FUNCTION_BLOCK FB_LinkedList_Test EXTENDS FB_TestSuite
VAR
END_VAR

NewListHasLength0();
isEmptyReturnsTrueOnEmptyList();
AddFirstNode();
AddMultipleNodesSameType();
AddMultipleNodesDifferentTypes();
InsertAfterSuccessfully();
RemoveNodeSuccessfully();

METHOD AddFirstNode
VAR
	fbLinkedList : FB_LinkedList;
	
	value : INT := 1;
	getValue : INT;
	
	Actual1 : BOOL;
	Actual2 : UINT;
	Actual3 : INT;
	
	Expected1 : BOOL := FALSE;
	Expected2 : UINT := 1;
	Expected3 : INT := 1;
END_VAR
TEST('AddFirstNode');

fbLinkedList.addValue(value);

Actual1 := fbLinkedList.isEmpty();
AssertEquals(Expected := Expected1, Actual := Actual1, Message := 'isEmpty returns true after adding an item to the list');

Actual2 := fbLinkedList.Length;
AssertEquals(Expected := Expected2, Actual := Actual2, Message := 'Length is not equal to 1 after adding 1 node');

fbLinkedList.getValue(0,getValue);
Actual3 := getValue;
AssertEquals(Expected := Expected3, Actual := Actual3, Message := 'getValue did not return the expected value');

TEST_FINISHED();
END_METHOD

METHOD AddMultipleNodesDifferentTypes
VAR
	fbLinkedList: FB_LinkedList;
	
	intValue 		: INT 		:= 33;
	realValue 		: REAL		:= 3.123;
	stringValue 	: STRING 	:= 'Hello world!';
	
	getInt : INT;
	getReal : REAL;
	getString : STRING;
	
	actualint : INT;
	actualReal : REAL;
	actualString : STRING;
END_VAR
TEST('AddMultipleNodesDifferentTypes');

fbLinkedList.addValue(intValue);
fbLinkedList.addValue(realValue);
fbLinkedList.addValue(stringValue);

fbLinkedList.getValue(0,getInt);
actualInt :=  getInt;
fbLinkedList.getValue(1, getReal);
actualReal := getReal;
fbLinkedList.getValue(2,getString);
actualString := getString;

AssertEquals_INT(expected := intValue, actual := actualInt, message := 'Position 0 was unexpected value');
AssertEquals_REAL(expected := realValue, actual := actualReal, delta := 0.01, message := 'Position 1 was unexpected value');
AssertEquals_STRING(expected := stringValue, actual := actualString, message := 'Position 2 was unexpceted value');

TEST_FINISHED();
END_METHOD

METHOD AddMultipleNodesSameType
VAR
	fbLinkedList : FB_LinkedList;
	intArray : ARRAY [0..4] OF INT := [1,2,3,4,5];
	i : INT;
	Actual: INT;
	ActualArr: INT;
	Expected: INT := 5;
	ExpectedArr: INT;
END_VAR
TEST('AddMultipleNodesSameType');

FOR i := 0 TO 4 DO
	fbLinkedList.addValue(intArray[i]);
END_FOR

Actual := fbLinkedList.Length;
AssertEquals(Expected := Expected, Actual := Actual, Message := 'Length not equal to 5 after adding 5 nodes');

FOR i := 0 TO 4 DO 
	fbLinkedList.getValue(i, ActualArr);
	ExpectedArr := intArray[i];
	AssertEquals(Expected := ExpectedArr, 
				 Actual := ActualArr, 
				 Message := CONCAT('Index ',CONCAT( INT_TO_STRING(i), CONCAT( ', expected ', CONCAT(INT_TO_STRING(ExpectedArr), CONCAT(', got ', INT_TO_STRING(ActualArr)))))));  
END_FOR

TEST_FINISHED();
END_METHOD

METHOD InsertAfterSuccessfully
VAR
	fbLinkedList : FB_LinkedList;
	initArray : ARRAY [0..4] OF INT := [1,2,3,4,5];
	i : INT;
	
	value : INT := 6;
	
	expectedArray : ARRAY [0..5] OF INT := [1,2,3,4,6,5];
	
	actual : INT;
	expected : INT;
END_VAR
TEST('InsertAfterSuccessfully');

FOR i := 0 TO 4 DO
	fbLinkedList.addValue(initArray[i]);
END_FOR

fbLinkedList.insertAfter(value, 3);

FOR i := 0 TO 4 DO 
	fbLinkedList.getValue(i, actual);
	expected := expectedArray[i];
	AssertEquals(Expected := Expected, Actual := Actual, Message := CONCAT('Index ', CONCAT(INT_TO_STRING(i), ' is not the expcted value'))); 
END_FOR

TEST_FINISHED();
END_METHOD

METHOD isEmptyReturnsTrueOnEmptyList
VAR
	fbLinkedList : FB_LinkedList;
	Expected : BOOL := TRUE;
	Actual: BOOL;
END_VAR
TEST('isEmptyReturnsTrueOnEmptyList');

Actual := fbLinkedList.isEmpty();

AssertEquals(Expected := Expected,
			 Actual := Actual,
			 Message := 'isEmpty() evaluates false on new linked list');
			 
TEST_FINISHED();
END_METHOD

METHOD NewListHasLength0
VAR
	LinkedList : FB_LinkedList;
	Result : UINT;
	ExpectedLength : UINT := 0;
END_VAR
TEST('NewListHasLength0');

Result := LinkedList.Length;

AssertEquals(Expected := ExpectedLength,
			Actual := Result,
			Message := 'New list is not empty');
			
			
	

TEST_FINISHED();
END_METHOD

METHOD RemoveNodeSuccessfully
VAR
	fbLinkedList : FB_LinkedList;
	initArray : ARRAY [0..4] OF INT := [1,2,3,4,5];
	i : INT;
	
	expectedArray : ARRAY [0..3] OF INT := [1,2,4,5];
	
	actual : INT;
	expected : INT;
END_VAR
TEST('RemoveNodeSuccessfully');

FOR i := 0 TO 4 DO
	fbLinkedList.addValue(initArray[i]);
END_FOR

fbLinkedList.remove(2);

FOR i := 0 TO 4 DO 
	fbLinkedList.getValue(i, actual);
	expected := expectedArray[i];
	AssertEquals(Expected := Expected, Actual := Actual, Message := CONCAT('Index ', CONCAT(INT_TO_STRING(i), ' is not the expcted value'))); 
END_FOR

TEST_FINISHED();
END_METHOD

END_FUNCTION_BLOCK

(* stored: Version 1.1.0.1
   POU FB_LinkedList_Test: Id {3d9ebd70-657f-405b-b31e-010edd5810ad}, SpecialFunc None
   Method AddFirstNode: Id {02c4374d-54e1-4c6d-a171-b7c57fceb053}
   Method AddMultipleNodesDifferentTypes: Id {cd39a802-fd8b-4efc-aea3-df781ae0ac28}
   Method AddMultipleNodesSameType: Id {8224b165-2d73-4654-aee9-e1a98ae56ad8}
   Method InsertAfterSuccessfully: Id {b32a3f05-51de-4288-b235-a3ce606ef510}
   Method isEmptyReturnsTrueOnEmptyList: Id {f9b33b21-fb22-40ad-9f99-3999b9a82141}
   Method NewListHasLength0: Id {4603ff7b-7599-41c0-8254-71412deb3ba7}
   Method RemoveNodeSuccessfully: Id {c44f33bf-39e0-48c8-bc35-5b1c8068d79a} *)
